(* IEC 61131-3 sources: DemoPumpStation/PumpStation/adapters, 5 files *)

(* ---- drive_adapter.st ---- *)
class DriveAdapter implements IPumpVfdDriveAdapter

var
    lastAction : string;
    vfdFrequency : lreal;
    state : VfdState := VfdState#stopped;
end_var

method public assignToVfd
var_input unitId : int; end_var
    lastAction := 'assign VFD';
    vfdFrequency := 45.0;
    state := VfdState#running;
end_method

method public transferToBypass
var_input unitId : int; end_var
    lastAction := 'to bypass';
    vfdFrequency := 45.0;
    state := VfdState#running;
end_method

method public stopUnit
var_input unitId : int; end_var
    lastAction := 'stop';

    // for demo simplicity
    vfdFrequency := 0.0;
    state := VfdState#stopped;
end_method

method public getVfdFrequency : lreal
    getVfdFrequency := vfdFrequency;
end_method

method public getVfdStatus : VfdState
    getVfdStatus := state;
end_method

end_class

(* ---- logger.st ---- *)
class TerminalLogger implements ILogger

var
    last : string;
end_var

method public info
var_input msg : string; end_var
    last := msg;
    __carrier_invoke('support.printf', 'Pump logger: %', msg);
end_method

end_class

(* ---- modbus_scada.st ---- *)
class PumpModbus implements IScadaModbus

var private
    modbus : Modbus.ModbusService;
    holdings, inputs : Modbus.ModbusSegment;
    notifier : Modbus.EmptyNotifier;
end_var

method public init
	var_input
	    settings_segment : ref_to array [*] of word;
    	feedback_segment : ref_to array [*] of word;
	end_var

	holdings.attachReadable('mbs', Modbus.ModbusArea#holds, 0, settings_segment);
	holdings.setRefreshMode(Modbus.ModbusRefreshMode#cyclic);

	inputs.attachWritable('mbs', Modbus.ModbusArea#inputs, 0, feedback_segment);
	inputs.setRefreshMode(Modbus.ModbusRefreshMode#cyclic);

	modbus.register(holdings);
	modbus.register(inputs);

	holdings.setNotifier(notifier);
	inputs.setNotifier(notifier);

end_method

method public process_pdi
var_in_out pdi : PumpStationControl; end_var
var
	codec : PdiCodec;
end_var
	codec.init(0, holdings);
	codec.decode(pdi);
end_method

method public process_pdo
var_input
	ctrl_state : PumpControllerViewModel;
	pumps_state : ref_to array[*] of PumpUnitView;
end_var
var
	codec : PdoCodec;
	i : udint;
end_var
	codec.init(0, inputs);

	codec.encode(ctrl_state);
	for i := lower_bound(pumps_state, 1)
				to upper_bound(pumps_state, 1) do codec.encode(ref(pumps_state^[i]));
	end_for

	inputs.publish();
end_method

method public iterate
	modbus.process();
end_method

end_class

(* ---- plc_info.st ---- *)
class LoopControl

var public
	task_id : string;
	period, old_start : lint;
end_var

var private
	main_dur : lint;
	last_end, last_start : lint;
end_var

	method private get_task_finish : lint
	var
		res : dint;
		dur : lint;
	end_var
		res := __carrier_invoke('sys.get_task_finish_time', task_id, ref(dur));
		if res = 0 then
			get_task_finish := dur;
		end_if
	end_method

	method private get_task_duration : lint
	var
		res : dint;
		dur : lint;
	end_var
		res := __carrier_invoke('sys.get_task_duration', task_id, ref(dur));
		if res = 0 then
			get_task_duration := dur;
		end_if
	end_method

	method public get_period
		main_dur := this.get_task_duration();
		last_end := this.get_task_finish();
		last_start := last_end - main_dur;

		period := last_start - old_start;
		old_start := last_start;
	end_method

end_class

(* ---- scada_presenter.st ---- *)
class BasicPumpStationPresenter implements IPumpStationPresenter

var
    drives : IPumpVfdDriveAdapter;
end_var

method public init
var_input d : IPumpVfdDriveAdapter; end_var
    drives := d;
end_method

method public buildView : PumpStationViewModel
var_input controller : ref_to PumpStationController; end_var

var
    vm : PumpStationViewModel;
    i : int;
end_var

    vm.isStarted := controller^.isStarted();
    vm.requestedUnits := controller^.getRequestedUnits();
    vm.activeUnits := controller^.getActiveUnits();

    vm.vfdUnitId := controller^.getVfdUnitId();
    vm.vfdFrequency := drives.getVfdFrequency();
    vm.vfdStatus := drives.getVfdStatus();

    for i := 1 to 4 do
        vm.pumps[i].id := int_to_uint(i);
        vm.pumps[i].role := controller^.getUnitRole(int_to_uint(i));
        vm.pumps[i].available := controller^.getUnitAvailable(int_to_uint(i));
        vm.pumps[i].faulted := controller^.getUnitFaulted(int_to_uint(i));
        vm.pumps[i].active := controller^.getUnitActive(int_to_uint(i));
    end_for

    buildView := vm;
end_method

end_class
